TYPE ECnv_Control_DUT :
STRUCT
	Mode:	UINT;
	Error:	BOOL;
	Warning:	UINT;
	Enabled:	BOOL;
	Stopped:	BOOL;
	Done:	BOOL;
	Running:	BOOL;
	Ready_For_Task:	BOOL;
	Current_Task_Type:	UINT;
	Current_Task_ID:	UINT;
	Cnv_Occupied:	BOOL;
	SM_State:	UINT;
	Motor:	Cnv_Motor_DUT;
	Instruction:	Cnv_Instruction_DUT;
	Inputs:	Cnv_Inputs_DUT;
	Cnv_Errors:	Cnv_Errors_DUT;
END_STRUCT
END_TYPE

(* stored: Version 1.1.0.1
   DUT ECnv_Control_DUT: Id {bd923e1c-5725-42ee-8a38-3f2c3f9e6c12} *)
